FUNCTION_BLOCK PUBLIC NidicIntegratedAxis_FB EXTENDS CoE_BasicAxis_FB  
VAR_INPUT		
		
END_VAR
VAR_IN_OUT	
END_VAR
VAR_OUTPUT	
END_VAR

VAR
	DebugError					: UINT;
	
END_VAR


AxisCtrlPtr^.Input.Parameter.Drive.eDriveType := enumDriveType.eIntegratedNidec;	
AxisCtrlPtr^.Input.Parameter.Drive.VendorNameID := eVendorNameID.Nidec;	
SUPER^(AxisRef:=AxisRef);

AxisCtrlPtr^.Output.Status.DriveEnable			:= io_StatusWord.4 AND  (io_StatusWord.0) ;	// DS-402 Status word bit 0 = Ready to switch on

METHOD CreateDriveErrMsgDetails : enumMotorEvents
VAR_INPUT
	ErrorId			: UDINT;
END_VAR

CASE ErrorId OF
	
	16#0:
		CreateDriveErrMsgDetails := enumMotorEvents.NoEvents;
		fnLogMsg(ADR(LogMsg_0),LOG_ERROR,'NidicInt Drive ErrorId %d  ,No error',UDINT_TO_DINT(ErrorId),0,0);
	16#2220:
		CreateDriveErrMsgDetails := enumMotorEvents.MotorSupplyError ;
		fnLogMsg(ADR(LogMsg_0),LOG_ERROR,'NidicInt Drive ErrorId %d Current, device outputside',UDINT_TO_DINT(ErrorId),0,0);	
	16#2250:
		CreateDriveErrMsgDetails := enumMotorEvents.MotorSupplyError ;
		fnLogMsg(ADR(LogMsg_0),LOG_ERROR,'NidicInt Drive ErrorId %d Short circuit/ground leakage',UDINT_TO_DINT(ErrorId),0,0);	

	16#2351:
		CreateDriveErrMsgDetails := enumMotorEvents.MotorSupplyError ;
		fnLogMsg(ADR(LogMsg_0),LOG_ERROR,'I2T THERMAL STATE LOAD EVEL WARNING',UDINT_TO_DINT(ErrorId),0,0);	
	
		
	16#3130:
		CreateDriveErrMsgDetails := enumMotorEvents.MotorSupplyError ;
		fnLogMsg(ADR(LogMsg_0),LOG_ERROR,'NidicInt Drive ErrorId %d Phase failure',UDINT_TO_DINT(ErrorId),0,0);
	
	16#3131:
		CreateDriveErrMsgDetails := enumMotorEvents.MotorSupplyError ;
		fnLogMsg(ADR(LogMsg_0),LOG_ERROR,'NidicInt Drive ErrorId %d Phase 1 failure',UDINT_TO_DINT(ErrorId),0,0);	

	16#3132:
		CreateDriveErrMsgDetails := enumMotorEvents.MotorSupplyError ;
		fnLogMsg(ADR(LogMsg_0),LOG_ERROR,'NidicInt Drive ErrorId %d Phase 2 failure',UDINT_TO_DINT(ErrorId),0,0);	
	
	16#3133:
		CreateDriveErrMsgDetails := enumMotorEvents.MotorSupplyError ;
		fnLogMsg(ADR(LogMsg_0),LOG_ERROR,'NidicInt Drive ErrorId %d Phase 3 failure',UDINT_TO_DINT(ErrorId),0,0);	
	

	16#3210:
		CreateDriveErrMsgDetails := enumMotorEvents.MotorSupplyError ;
		fnLogMsg(ADR(LogMsg_0),LOG_ERROR,'NidicInt Drive ErrorId %d DC link over-voltage',UDINT_TO_DINT(ErrorId),0,0);	

		 
	16#3220:
		CreateDriveErrMsgDetails := enumMotorEvents.MotorSupplyError; 
		fnLogMsg(ADR(LogMsg_0),LOG_ERROR,'NidicInt Drive ErrorId %d DC Link under voltage',UDINT_TO_DINT(ErrorId),0,0);
	
	16#3331:
		CreateDriveErrMsgDetails := enumMotorEvents.MotorSupplyError; 
		fnLogMsg(ADR(LogMsg_0),LOG_ERROR,'NidicInt Drive ErrorId %d FIELD CIRCUIT INTERRUPTED',UDINT_TO_DINT(ErrorId),0,0);
	
	
	16#4210:
		CreateDriveErrMsgDetails := enumMotorEvents.MotorOverTemp; 
		fnLogMsg(ADR(LogMsg_0),LOG_ERROR,'NidicInt Drive ErrorId %d Excess temperature drive',UDINT_TO_DINT(ErrorId),0,0);
		
	16#4310:
		CreateDriveErrMsgDetails := enumMotorEvents.MotorOverTemp; 
		fnLogMsg(ADR(LogMsg_0),LOG_ERROR,'NidicInt Drive ErrorId %d Excess temperature device',UDINT_TO_DINT(ErrorId),0,0);		
		

	16#5300:
		 CreateDriveErrMsgDetails := enumMotorEvents.MotorGeneralError;
		 fnLogMsg(ADR(LogMsg_0),LOG_ERROR,'NidicInt Drive ErrorId %d Control device hardware',UDINT_TO_DINT(ErrorId),0,0);

	16#6010:
		CreateDriveErrMsgDetails := enumMotorEvents.MotorGeneralError;
 		fnLogMsg(ADR(LogMsg_0),LOG_ERROR, 'NidicInt Drive ErrorId %d Software reset',UDINT_TO_DINT(ErrorId),0,0);

	16#6320:
		CreateDriveErrMsgDetails := enumMotorEvents.PLCIllegalParam; 
		fnLogMsg(ADR(LogMsg_0),LOG_ERROR,'NidicInt Drive ErrorId %d Parameter Error',UDINT_TO_DINT(ErrorId),0,0);


(*chopper 10 - Th Brake Res*)

	16#7121:
		CreateDriveErrMsgDetails := enumMotorEvents.MotorStalled; 
		fnLogMsg(ADR(LogMsg_0),LOG_ERROR,'NidicInt Drive ErrorId %d  Motor error OR commutation malfunction',UDINT_TO_DINT(ErrorId),0,0);
	16#7300:
		CreateDriveErrMsgDetails := enumMotorEvents.MotorFeedBackErr; 
		fnLogMsg(ADR(LogMsg_0),LOG_ERROR, 'NidicInt Drive ErrorId %d Sensor Error',UDINT_TO_DINT(ErrorId),0,0);

	16#7500:
		CreateDriveErrMsgDetails := enumMotorEvents.DriveComError; 
		fnLogMsg(ADR(LogMsg_0),LOG_ERROR,'NidicInt Drive ErrorId %d Communication 90 - Power Comms',UDINT_TO_DINT(ErrorId),0,0);

	
		
	ELSE
		fnLogMsg(ADR(LogMsg_0),LOG_ERROR,'unknown NidicInt Drive ErrorId %d ',UDINT_TO_DINT(ErrorId),0,0);
		CreateDriveErrMsgDetails := enumMotorEvents.NoEvents;
	END_CASE
END_METHOD

METHOD  INIT_Specific : BOOL 
VAR_INPUT
	bStart: 					BOOL;
END_VAR
VAR_INST	
	ComDelay:	TON;
	Nidec_Init_State : INT ;
	ExecuteTrig: 	Trigger;
END_VAR
IF ExecuteTrig.EDGEPOS(bStart) THEN
	INIT_Specific := FALSE ;
	IF AxisCtrlPtr^.Input.Parameter.Drive.bDisableFoE_Transfer THEN 
		Nidec_Init_State:= 5;//10;
	ELSE
		Nidec_Init_State:= 1;
	END_IF
END_IF


IF ExecuteTrig.EDGENEG(bStart) THEN
	Nidec_Init_State := 0;
END_IF	

	
CASE Nidec_Init_State OF							
						
	1:	
		Nidec_Init_State:= 5;			
	5:
		ReadInitDriveParID(FALSE);
		Nidec_Init_State:=	6;
		
	6:
		IF ReadInitDriveParID(TRUE) THEN
			Nidec_Init_State:=	10;
		END_IF
	
	
	10:
		
		Nidec_Init_State := 0 ;
		INIT_Specific := TRUE ;
		AxisCtrlPtr^.Output.Status.AxisInitDone := TRUE ;
		AxisCtrlPtr^.Output.Status.ReadyForCmd := TRUE ;
END_CASE
END_METHOD

METHOD ReadInitDriveParID : BOOL
VAR_INPUT
	bStart : BOOL;
END_VAR

VAR_INST
	ExecuteTrig_1: 		Trigger;
	State_InitSpecific_1: INT;
END_VAR

IF ExecuteTrig_1.EDGEPOS(bStart) THEN
	ReadInitDriveParID		:= FALSE;
	State_InitSpecific_1	:= 1;		
END_IF

IF ExecuteTrig_1.EDGENEG(bStart) THEN
	State_InitSpecific_1	:= 0;	
	ReadInitDriveParID		:= FALSE;
END_IF

CASE State_InitSpecific_1 OF

	0:
	
	1:
		SUPER^.EcCoeSdoRead(FALSE);
		CoeSdoRW.Input.Read.nIndex		:= DINT_TO_WORD(eNidecDriveParID.Menue05);
		CoeSdoRW.Input.Read.nSubIndex	:= 7;
		CoeSdoRW.Input.Read.pDstBuf		:= ADR(CoeRead_RatedCurrent);
		CoeSdoRW.Input.Read.cbBufLen	:= SIZEOF(CoeRead_RatedCurrent);
		State_InitSpecific_1	:= 2;
		
	2:
		IF SUPER^.EcCoeSdoRead(TRUE) THEN	
			State_InitSpecific_1	:= 3;
		END_IF
		
	3:
		SUPER^.EcCoeSdoRead(FALSE);
		CoeSdoRW.Input.Read.nIndex		:= DINT_TO_WORD(eNidecDriveParID.Menue04);
		CoeSdoRW.Input.Read.nSubIndex	:= 41;
		CoeSdoRW.Input.Read.pDstBuf		:= ADR(CoeRead_RatedTorque);
		CoeSdoRW.Input.Read.cbBufLen	:= SIZEOF(CoeRead_RatedTorque);
		State_InitSpecific_1	:= 4;
		
	4:
		IF SUPER^.EcCoeSdoRead(TRUE) THEN
			AxisCtrlPtr^.Input.Parameter.RatedCurrent	:= UDINT_TO_LREAL(CoeRead_RatedCurrent) / 1000.0;
			AxisCtrlPtr^.Input.Parameter.Ratedtorque	:= UDINT_TO_LREAL(CoeRead_RatedTorque) / 100.0;
			ReadInitDriveParID		:= TRUE;	
			State_InitSpecific_1	:= 0;
		END_IF
		
		
 
		
END_CASE
END_METHOD

END_FUNCTION_BLOCK

(* stored: Version 1.1.0.1, ProductVersion 3.1.4024.3
   POU NidicIntegratedAxis_FB: Id {7e38e8dc-2963-4430-8373-393f639f57b8}, SpecialFunc None
   Method CreateDriveErrMsgDetails: Id {deb186b6-70ae-43b0-9cbd-328800775daf}
   Method INIT_Specific: Id {7498f1be-e9ec-49c9-9517-b374b5129cd3}
   Method ReadInitDriveParID: Id {f41d77ab-ecc7-4731-be6e-6c6802960626} *)
